TYPE EXAMPLEJSONSTRUCT :
STRUCT
	var1: JSONVAR;
	var2: JSONVAR;
	var3: JSONVAR;
	obj: EXAMPLEJSONSTRUCT_1;
	arrayobj: ARRAY[1..3] OF JSONVAR;
END_STRUCT
END_TYPE

(* stored: Version 1.1.0.1
   DUT EXAMPLEJSONSTRUCT: Id {535e1966-3fb6-4089-bf5a-f928340d1f23} *)
